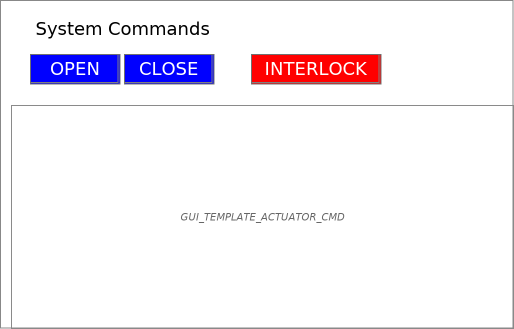
VISUALIZATION GUI_PVV1_CMD  // 514x329
    Frame (11,105 503x224)
        shows GUI_TEMPLATE_ACTUATOR_CMD(m_Instance := MAIN.cmdPVV1)
    Button (30,54 90x30), "OPEN", tooltip "Set External System command to OPEN"
        OnMouseClick: execute { MAIN.bCmdPVV1 := TRUE; }
    Button (124,54 90x30), "CLOSE", tooltip "Set External System command to CLOSE"
        OnMouseClick: execute { MAIN.bCmdPVV1 := FALSE; }
    Rectangle (33,14 180x30), "System Commands"
    Button (251,54 130x30), "INTERLOCK", tooltip "Toggle External System INTERLOCK"
        toggle MAIN.bIntlkPVV1
        OnMouseClick: execute { MAIN.bCmdPVV1 := TRUE; }
END_VISUALIZATION

(* stored: Version 1.1.0.1, ProductVersion 3.1.4024.9
   Visu GUI_PVV1_CMD: Id {86d18cca-61a5-4a00-b3cd-5b98ff245187} *)
